{attribute 'linkalways'} 
{attribute 'no_explicit_call' := 'This FB is a CLASS and must be accessed using methods or properties'}
{attribute 'enable_dynamic_creation'}
FUNCTION_BLOCK Session EXTENDS Disposable IMPLEMENTS I_Session
VAR
	_id : T_MAXSTRING;
	_lastAccessedTimestamp : SystemTimestamp;
	sessionStorage : Dictionary;
END_VAR

METHOD PUBLIC AddOrUpdateStorage
VAR_INPUT
	StorageId : T_MAXSTRING;
	Source : I_SessionData;
END_VAR
sessionStorage.AddOrUpdate(StorageId, Source);
END_METHOD

METHOD PUBLIC DisposeAllDataFromStorage
VAR_INPUT
END_VAR
VAR
	enumerator : I_ForwardEnumerator;
	sessionData : I_SessionData;
END_VAR
enumerator := sessionStorage.GetEnumerator();

WHILE enumerator.MoveNext() DO
	IF enumerator.TryGet(sessionData) THEN
		sessionData.Dispose();
	END_IF
END_WHILE

enumerator.Dispose();
sessionStorage.Clear();
END_METHOD

METHOD PUBLIC DisposeDataFromStorage
VAR_INPUT
	StorageId : T_MAXSTRING;
END_VAR
VAR
	sessionData : I_SessionData;
END_VAR
IF NOT sessionStorage.TryGetValue(StorageId,sessionData) THEN
	RETURN;
END_IF

sessionData.Dispose();
sessionStorage.Remove(StorageId);
END_METHOD

METHOD FB_exit : BOOL
VAR_INPUT
	bInCopyCode : BOOL; // if TRUE, the exit method is called for exiting an instance that is copied afterwards (online change).
END_VAR
IF bInCopyCode THEN
	RETURN;
END_IF

DisposeAllDataFromStorage();
END_METHOD

METHOD FB_init : BOOL
VAR_INPUT
	bInitRetains : BOOL; // if TRUE, the retain variables are initialized (warm start / cold start)
	bInCopyCode : BOOL;  // if TRUE, the instance afterwards gets moved into the copy code (online change)
	SessionId : T_MAXSTRING;
END_VAR
_id := SessionId;
END_METHOD

PROPERTY PUBLIC Id : T_MAXSTRING
GET
Id := _id;
END_GET
END_PROPERTY

PROPERTY PUBLIC LastAccessedTimestamp : I_TimeStamp
GET
LastAccessedTimestamp := _lastAccessedTimestamp;
END_GET
END_PROPERTY

METHOD PUBLIC Refresh
VAR_INPUT
END_VAR
_lastAccessedTimestamp.SetNow();
END_METHOD

METHOD PUBLIC TryGetDataFromStorage : BOOL
VAR_INPUT
	StorageId : T_MAXSTRING;
	Destination : REFERENCE TO I_SessionData;
END_VAR
TryGetDataFromStorage := sessionStorage.TryGetValue(StorageId, Destination);
END_METHOD

END_FUNCTION_BLOCK

(* stored: Version 1.1.0.1, ProductVersion 3.1.4024.12
   POU Session: Id {92b2871e-981c-401e-a212-a2d1d9c07815}, SpecialFunc None
   Folder Constructor: Id {8592cdb5-cda5-4488-a7d8-7f9298e4c6eb}
   Folder Destructor: Id {fb318f0b-2e08-4568-af7e-b120b123a70c}
   Method AddOrUpdateStorage: Id {e26f978d-d270-4745-b672-d6bde43eb40d}
   Method DisposeAllDataFromStorage: Id {17ac81c5-d932-41ed-ab94-5a3293696a05}
   Method DisposeDataFromStorage: Id {61bc8675-9d6b-4fe1-9662-439e29934dc1}
   Method FB_exit: Id {9d0a64cf-8f69-4161-914e-ccc4710673a9}
   Method FB_init: Id {8e5729a5-989c-4b7b-be1c-46f3a4b580a7}
   Property Id: Id {baad7f6b-69c2-485f-a2ea-9fcac8d9766e}
   Get Get: Id {b76e7d95-4e69-41b2-98af-d8efaa8e87c3}
   Property LastAccessedTimestamp: Id {4cfbcf71-6e77-4d73-a567-8c951de8c083}
   Get Get: Id {3b6c2e8e-3487-49f8-8112-6e416aa1be0d}
   Method Refresh: Id {9813f788-a2ed-4ed5-bd00-5b6f69a81564}
   Method TryGetDataFromStorage: Id {490aeb08-e407-49ba-8054-c25284551ce2} *)
